// LS Electric XG5000 project: 91
// PLC NewPLC
// module base 0 slot 0: 입출력 모듈:XBC-DN/DP14E (DC 24V 입력 8점, 트랜지스터 출력 6점)

PROGRAM NewProgram (task: 스캔 프로그램)

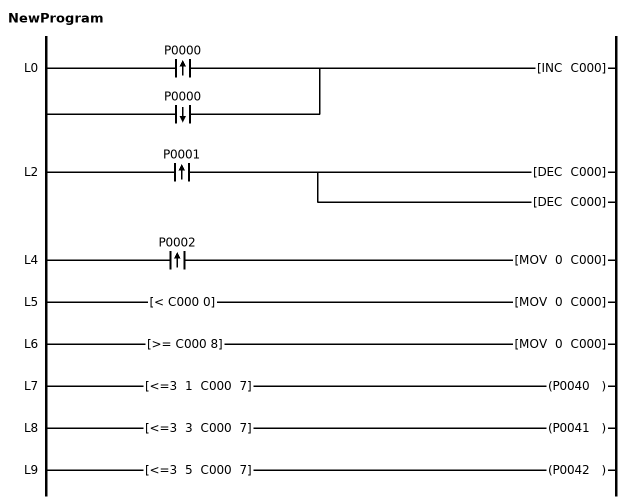
; L0
LOADP     P0000
ORN       P0000
INC       C000
; L2
LOADP     P0001
DEC       C000
DEC       C000
; L4
LOADP     P0002
MOV       0 C000
; L5
LOAD<     C000 0
MOV       0 C000
; L6
LOAD>=    C000 8
MOV       0 C000
; L7
LOAD<=3   1 C000 7
OUT       P0040
; L8
LOAD<=3   3 C000 7
OUT       P0041
; L9
LOAD<=3   5 C000 7
OUT       P0042